FUNCTION_BLOCK FB_Station_LowerZForce EXTENDS FB_CH_Object
VAR
	ipStation : I_XP_Station_PLC;
	nSeq : UINT;
	fbTon : TON;
	ipMoverInStation : I_XP_Mover_PLC;
	bFromUpstreamProcessIsFinish: BOOL := TRUE;
	sTargetStation : STRING; //the mover gets this as next target
END_VAR

METHOD FB_init : BOOL
VAR_INPUT
	bInitRetains : BOOL; // if TRUE, the retain variables are initialized (warm start / cold start)
	bInCopyCode : BOOL;  // if TRUE, the instance afterwards gets moved into the copy code (online change)
	
	ipStation : I_XP_Station_PLC;
	
END_VAR
VAR
	fbGetCurTaskIdx  : GETCURTASKINDEX;
END_VAR
THIS^.ipStation := ipStation;
END_METHOD

{attribute 'monitoring':='call'}
 //the mover gets this as next target
PROPERTY TargetStation : STRING
GET
TargetStation := sTargetStation;
END_GET
SET
sTargetStation := TargetStation;
END_SET
END_PROPERTY

METHOD Update : HRESULT
VAR
	refPlanarTrack : REFERENCE TO MC_PlanarTrack;
END_VAR
IF ipStation = 0 THEN
	RETURN; // ERROR
END_IF

IF ipStation.System.Disabled THEN
	nSeq := 0;
END_IF

//The simulation (automatic retransmission of a mover after a fixed time) is stopped for this station
ipStation.SimulationStop();

CASE nSeq OF 

	0: //wait for mover
		IF ipStation.MoversInPlace THEN
			//receive the foremost mover in the station (if there is more than one mover in the station)
			ipMoverInStation := ipStation.MoversInQueue[0];
			nSeq := 1;
		END_IF
		
	1: //Z = 0
		ipMoverInStation.LowerToUnknownLevel();
		nSeq := 2;				

	2: // wait until lowering is finish
		IF ipMoverInStation.Feedback.Done THEN
			fbTon.IN := FALSE;
			nSeq := 3;	
		END_IF
		
	3: //Delay 5s
		fbTon.IN := TRUE;
		IF fbTon.q THEN
			nSeq := 4;	
		END_IF			

	4: //Lift
		ipMoverInStation.LiftFromUnknownLevel();
		nSeq := 5;				

	5: // wait until lifting is finish
		//The upstream process can set this bool if the process is finish and the mover can leave the station
		bFromUpstreamProcessIsFinish := bFromUpstreamProcessIsFinish;

		fbTon.IN := TRUE;
		IF fbTon.q AND bFromUpstreamProcessIsFinish THEN
			nSeq := 100;	
		END_IF

		
	100: // send movers away to next target station or groupe. If no target exist, wait in this step
		IF sTargetStation <> '' THEN
			ipStation.SendMoversToStation(THIS^.sTargetStation);
			nSeq := 0;	
		END_IF

	
END_CASE
fbTon(PT:= T#5S);
END_METHOD

END_FUNCTION_BLOCK

(* stored: Version 1.1.0.1, ProductVersion 3.1.4026.12
   POU FB_Station_LowerZForce: Id {986f1d68-bf8e-4783-9c03-c01052f5acdc}, SpecialFunc None
   Method FB_init: Id {4337220f-62bf-48d1-af24-ba632db2ff2c}
   Property TargetStation: Id {b8475f86-11ac-454e-bb60-686b1712227c}
   Get Get: Id {5d579e06-88ee-4aa6-a2fa-7633fd86f1fb}
   Set Set: Id {836bf01a-e060-4d8a-9635-cf3dd29b47a6}
   Method Update: Id {dc7ca279-7959-4b33-8e61-bcdf95f8089d} *)
